// TwinCAT 3 PLC project GmdPlc
// ProgramVersion: 3.1.4022.3
// libraries:
//   L2SI Vacuum Library, * (SLAC)
//   LCLS General, * (SLAC)
//   Tc2_Standard, * (Beckhoff Automation GmbH)
//   Tc2_System, * (Beckhoff Automation GmbH)
//   Tc2_Utilities, * (Beckhoff Automation GmbH)
//   Tc3_Module, * (Beckhoff Automation GmbH)
// project tree:
//   GVLs/ GVL_GMD.TcGVL, GVL_VARIABLES.TcGVL
//   / PlcTask.TcTTO
//   POUs/ MAIN.TcPOU, PRG_DIAGNOSTIC.TcPOU, PRG_GMD.TcPOU
// real-time tasks:
//   TASK PlcTask: cycle T#10ms, priority 20, ADS port 350
//   TASK SimTask: cycle T#5ms, priority 21, ADS port 351
// I/O:
//   DEVICE =+-EK1100_00_00-CPU/EtherCAT1, AmsNetId 5.56.6.154.2.1
//     =+-EK1100_00_00 [EK1100 EtherCAT Coupler (2A E-Bus)]
//       =+-EK1110_00_08 [EK1110 EtherCAT extension]
//     =+-EL3174-02_04_08 [EL3174 4Ch. Ana. Input +/-10V Diff., +/-20mA SingleEnded, 16 Bit]
//     =+-ES9187_02_13 [EL9187 Potential Connection, 8 x Ground]
//     =+-ES9187_02_09 [EL9187 Potential Connection, 8 x Ground]
//     =+-ES9187_01_13 [EL9187 Potential Connection, 8 x Ground]
//     =+-ES9187_01_08 [EL9187 Potential Connection, 8 x Ground]
//     =+-ES9187_01_03 [EL9187 Potential Connection, 8 x Ground]
//     =+-ES9184_04_14 [EL9184 Potential Connection, 8 x 24V, 8 x Ground]
//     =+-ES9184_00_05 [EL9184 Potential Connection, 8 x 24V, 8 x Ground]
//     =+-ES9070_04_12 [EL9070 Shield terminal]
//     =+-ES9070_04_09 [EL9070 Shield terminal]
//     =+-ES9070_04_04 [EL9070 Shield terminal]
//     =+-ES9070_00_03 [EL9070 Shield terminal]
//     =+-ES7041_04_01 [EL7041 1Ch. Stepper motor output stage (50V, 5A)]
//     =+-ES4004_04_05 [EL4004 4Ch. Ana. Output 0-10V, 12bit]
//     =+-ES3202_04_10 [EL3202 2Ch. Ana. Input PT100 (RTD)]
//     =+-ES3068_01_14 [EL3068 8Ch. Ana. Input 0-10V]
//     =+-ES3068_01_12 [EL3068 8Ch. Ana. Input 0-10V]
//     =+-ES3068_01_09 [EL3068 8Ch. Ana. Input 0-10V]
//     =+-ES3068_01_07 [EL3068 8Ch. Ana. Input 0-10V]
//     =+-ES3068_01_04 [EL3068 8Ch. Ana. Input 0-10V]
//     =+-ES3068_01_02 [EL3068 8Ch. Ana. Input 0-10V]
//     =+-ES3064_04_11 [EL3064 4Ch. Ana. Input 0-10V]
//     =+-ES3064_00_02 [EL3064 4Ch. Ana. Input 0-10V]
//     =+-ES2088_02_14 [EL2088 8Ch. Dig. Output 24V, 0.5A, switching to negative]
//     =+-ES2088_02_10 [EL2088 8Ch. Dig. Output 24V, 0.5A, switching to negative]
//     =+-ES2008_04_15 [EL2008 8Ch. Dig. Output 24V, 0.5A]
//     =+-ES2008_00_06 [EL2008 8Ch. Dig. Output 24V, 0.5A]
//     =+-ES2004_04_07 [EL2004 4Ch. Dig. Output 24V, 0.5A]
//     =+-ES2004_04_06 [EL2004 4Ch. Dig. Output 24V, 0.5A]
//     =+-ES2004_02_05 [EL2004 4Ch. Dig. Output 24V, 0.5A]
//     =+-ES2004_02_02 [EL2004 4Ch. Dig. Output 24V, 0.5A]
//     =+-ES1088_02_15 [EL1088 8Ch. Dig. Input 24V, 3ms, negative]
//     =+-ES1088_02_12 [EL1088 8Ch. Dig. Input 24V, 3ms, negative]
//     =+-ES1088_02_11 [EL1088 8Ch. Dig. Input 24V, 3ms, negative]
//     =+-ES1088_02_08 [EL1088 8Ch. Dig. Input 24V, 3ms, negative]
//     =+-ES1008_04_13 [EL1008 8Ch. Dig. Input 24V, 3ms]
//     =+-ES1008_00_04 [EL1008 8Ch. Dig. Input 24V, 3ms]
//     =+-ES1004_02_06 [EL1004 4Ch. Dig. Input 24V, 3ms]
//     =+-ES1004_02_04 [EL1004 4Ch. Dig. Input 24V, 3ms]
//     =+-ES1004_02_03 [EL1004 4Ch. Dig. Input 24V, 3ms]
//     =+-ES1004_02_01 [EL1004 4Ch. Dig. Input 24V, 3ms]
//     =+-EL9400_02_07 [EL9400 E-Bus Power Supplier]
//     =+-EL2794_04_16 [EL2794 4Ch. Dig. Output 24V AC/DC, 2A, short-circuit-proof]
//     =+-EL2794_04_02 [EL2794 4Ch. Dig. Output 24V AC/DC, 2A, short-circuit-proof]
//     =+-EL2794_01_15 [EL2794 4Ch. Dig. Output 24V AC/DC, 2A, short-circuit-proof]
//     =+-EL2794_01_11 [EL2794 4Ch. Dig. Output 24V AC/DC, 2A, short-circuit-proof]
//     =+-EL2794_01_10 [EL2794 4Ch. Dig. Output 24V AC/DC, 2A, short-circuit-proof]
//     =+-EL2794_01_06 [EL2794 4Ch. Dig. Output 24V AC/DC, 2A, short-circuit-proof]
//     =+-EL2794_01_05 [EL2794 4Ch. Dig. Output 24V AC/DC, 2A, short-circuit-proof]
//     =+-EL2794_01_01 [EL2794 4Ch. Dig. Output 24V AC/DC, 2A, short-circuit-proof]
//     =+-EL2794_00_07 [EL2794 4Ch. Dig. Output 24V AC/DC, 2A, short-circuit-proof]
//     =+-EL1004_04_03 [EL1004 4Ch. Dig. Input 24V, 3ms]
//     =+-EK1110_04_17 [EK1110 EtherCAT extension]
//   DEVICE SimDevice 2 (EtherCAT Simulation), AmsNetId 5.45.6.154.3.1
//     =+-EK1100_00_00 // EK1100-0000-0018
//     =+-EK1110_00_08 // EK1110-0000-0017
//     =+-EL3174-02_04_08 // EL3174-0000-0016
//     =+-ES7041_04_01 // EL7041-0000-0025
//     =+-ES4004_04_05 // EL4004-0000-0020
//     =+-ES3202_04_10 // EL3202-0000-0022
//     =+-ES3068_01_14 // EL3068-0000-0020
//     =+-ES3068_01_12 // EL3068-0000-0020
//     =+-ES3068_01_09 // EL3068-0000-0020
//     =+-ES3068_01_07 // EL3068-0000-0020
//     =+-ES3068_01_04 // EL3068-0000-0020
//     =+-ES3068_01_02 // EL3068-0000-0020
//     =+-ES3064_04_11 // EL3064-0000-0020
//     =+-ES3064_00_02 // EL3064-0000-0020
//     =+-ES2088_02_14 // EL2088-0000-0018
//     =+-ES2088_02_10 // EL2088-0000-0018
//     =+-ES2008_04_15 // EL2008-0000-0018
//     =+-ES2008_00_06 // EL2008-0000-0018
//     =+-ES2004_04_07 // EL2004-0000-0018
//     =+-ES2004_04_06 // EL2004-0000-0018
//     =+-ES2004_02_05 // EL2004-0000-0018
//     =+-ES2004_02_02 // EL2004-0000-0018
//     =+-ES1088_02_15 // EL1088-0000-0018
//     =+-ES1088_02_12 // EL1088-0000-0018
//     =+-ES1088_02_11 // EL1088-0000-0018
//     =+-ES1088_02_08 // EL1088-0000-0018
//     =+-ES1008_04_13 // EL1008-0000-0018
//     =+-ES1008_00_04 // EL1008-0000-0018
//     =+-ES1004_02_06 // EL1004-0000-0019
//     =+-ES1004_02_04 // EL1004-0000-0019
//     =+-ES1004_02_03 // EL1004-0000-0019
//     =+-ES1004_02_01 // EL1004-0000-0019
//     =+-EL2794_04_16 // EL2794-0000-0016
//     =+-EL2794_04_02 // EL2794-0000-0016
//     =+-EL2794_01_15 // EL2794-0000-0016
//     =+-EL2794_01_11 // EL2794-0000-0016
//     =+-EL2794_01_10 // EL2794-0000-0016
//     =+-EL2794_01_06 // EL2794-0000-0016
//     =+-EL2794_01_05 // EL2794-0000-0016
//     =+-EL2794_01_01 // EL2794-0000-0016
//     =+-EL2794_00_07 // EL2794-0000-0016
//     =+-EL1004_04_03 // EL1004-0000-0019
//     =+-EK1110_04_17 // EK1110-0000-0017
// variable links:
//   GmdPlc/GmdPlc Instance <-> =+-EK1100_00_00-CPU/EtherCAT1/=+-EL1004_04_03
//     PlcTask Inputs/GVL_GMD.fb_EM1K0_GMD_PRT_40.i_xAlarmOK <-> Channel 2/Input
//     PlcTask Inputs/GVL_GMD.fb_EM1K0_GMD_PRT_40.i_xIsRun <-> Channel 1/Input
//   GmdPlc/GmdPlc Instance <-> =+-EK1100_00_00-CPU/EtherCAT1/=+-EL2794_01_01
//     PlcTask Outputs/GVL_GMD.fb_EM1K0_GMD_GCC_10.q_xHV_DIS <-> Channel 1/Output
//     PlcTask Outputs/GVL_GMD.fb_EM1K0_GMD_GCC_20.q_xHV_DIS <-> Channel 2/Output
//     PlcTask Outputs/GVL_GMD.fb_EM1K0_GMD_GCC_30.q_xHV_DIS <-> Channel 3/Output
//   GmdPlc/GmdPlc Instance <-> =+-EK1100_00_00-CPU/EtherCAT1/=+-EL2794_01_05
//     PlcTask Outputs/GVL_GMD.fb_EM1K0_GMD_GCC_40.q_xHV_DIS <-> Channel 2/Output
//   GmdPlc/GmdPlc Instance <-> =+-EK1100_00_00-CPU/EtherCAT1/=+-EL2794_01_06
//     PlcTask Outputs/GVL_GMD.fb_EM1K0_GMD_GCC_50.q_xHV_DIS <-> Channel 1/Output
//     PlcTask Outputs/GVL_GMD.fb_EM1K0_GMD_GCC_60.q_xHV_DIS <-> Channel 2/Output
//   GmdPlc/GmdPlc Instance <-> =+-EK1100_00_00-CPU/EtherCAT1/=+-EL2794_01_10
//     PlcTask Outputs/GVL_GMD.fb_EM1K0_GMD_GCC_70.q_xHV_DIS <-> Channel 1/Output
//   GmdPlc/GmdPlc Instance <-> =+-EK1100_00_00-CPU/EtherCAT1/=+-EL2794_04_02
//     PlcTask Outputs/GVL_GMD.fb_EM1K0_GMD_PRT_40.q_xRemote <-> Channel 2/Output
//     PlcTask Outputs/GVL_GMD.fb_EM1K0_GMD_PRT_40.q_xRunDo <-> Channel 1/Output
//   GmdPlc/GmdPlc Instance <-> =+-EK1100_00_00-CPU/EtherCAT1/=+-ES1004_02_01
//     PlcTask Inputs/GVL_GMD.fb_EM1K0_GMD_VRC_10.i_xClsLS <-> Channel 2/Input
//     PlcTask Inputs/GVL_GMD.fb_EM1K0_GMD_VRC_20.i_xClsLS <-> Channel 4/Input
//     PlcTask Inputs/GVL_GMD.fb_EM1K0_GMD_VRC_10.i_xOpnLS <-> Channel 1/Input
//     PlcTask Inputs/GVL_GMD.fb_EM1K0_GMD_VRC_20.i_xOpnLS <-> Channel 3/Input
//   GmdPlc/GmdPlc Instance <-> =+-EK1100_00_00-CPU/EtherCAT1/=+-ES1004_02_03
//     PlcTask Inputs/GVL_GMD.fb_EM1K0_GMD_VRC_30.i_xClsLS <-> Channel 2/Input
//     PlcTask Inputs/GVL_GMD.fb_EM1K0_GMD_VRC_30.i_xOpnLS <-> Channel 1/Input
//   GmdPlc/GmdPlc Instance <-> =+-EK1100_00_00-CPU/EtherCAT1/=+-ES1004_02_04
//     PlcTask Inputs/GVL_GMD.fb_EM1K0_GMD_VRC_50.i_xClsLS <-> Channel 2/Input
//     PlcTask Inputs/GVL_GMD.fb_EM1K0_GMD_VRC_60.i_xClsLS <-> Channel 4/Input
//     PlcTask Inputs/GVL_GMD.fb_EM1K0_GMD_VRC_50.i_xOpnLS <-> Channel 1/Input
//     PlcTask Inputs/GVL_GMD.fb_EM1K0_GMD_VRC_60.i_xOpnLS <-> Channel 3/Input
//   GmdPlc/GmdPlc Instance <-> =+-EK1100_00_00-CPU/EtherCAT1/=+-ES1004_02_06
//     PlcTask Inputs/GVL_GMD.fb_EM1K0_GMD_VRC_70.i_xClsLS <-> Channel 2/Input
//     PlcTask Inputs/GVL_GMD.fb_EM1K0_GMD_VRC_70.i_xOpnLS <-> Channel 1/Input
//   GmdPlc/GmdPlc Instance <-> =+-EK1100_00_00-CPU/EtherCAT1/=+-ES1088_02_08
//     PlcTask Inputs/GVL_GMD.fb_EM1K0_GMD_PTM_10.i_xAtSpd <-> Channel 1/Input
//     PlcTask Inputs/GVL_GMD.fb_EM1K0_GMD_PTM_20.i_xAtSpd <-> Channel 3/Input
//     PlcTask Inputs/GVL_GMD.fb_EM1K0_GMD_PTM_10.i_xFault <-> Channel 2/Input
//     PlcTask Inputs/GVL_GMD.fb_EM1K0_GMD_PTM_20.i_xFault <-> Channel 4/Input
//   GmdPlc/GmdPlc Instance <-> =+-EK1100_00_00-CPU/EtherCAT1/=+-ES1088_02_11
//     PlcTask Inputs/GVL_GMD.fb_EM1K0_GMD_PTM_30.i_xAtSpd <-> Channel 1/Input
//     PlcTask Inputs/GVL_GMD.fb_EM1K0_GMD_PTM_40.i_xAtSpd <-> Channel 3/Input
//     PlcTask Inputs/GVL_GMD.fb_EM1K0_GMD_PTM_30.i_xFault <-> Channel 2/Input
//     PlcTask Inputs/GVL_GMD.fb_EM1K0_GMD_PTM_40.i_xFault <-> Channel 4/Input
//   GmdPlc/GmdPlc Instance <-> =+-EK1100_00_00-CPU/EtherCAT1/=+-ES1088_02_12
//     PlcTask Inputs/GVL_GMD.fb_EM1K0_GMD_PTM_50.i_xAtSpd <-> Channel 1/Input
//     PlcTask Inputs/GVL_GMD.fb_EM1K0_GMD_PTM_60.i_xAtSpd <-> Channel 3/Input
//     PlcTask Inputs/GVL_GMD.fb_EM1K0_GMD_PTM_50.i_xFault <-> Channel 2/Input
//     PlcTask Inputs/GVL_GMD.fb_EM1K0_GMD_PTM_60.i_xFault <-> Channel 4/Input
//   GmdPlc/GmdPlc Instance <-> =+-EK1100_00_00-CPU/EtherCAT1/=+-ES1088_02_15
//     PlcTask Inputs/GVL_GMD.fb_EM1K0_GMD_PTM_70.i_xAtSpd <-> Channel 1/Input
//     PlcTask Inputs/GVL_GMD.fb_EM1K0_GMD_PTM_70.i_xFault <-> Channel 2/Input
//   GmdPlc/GmdPlc Instance <-> =+-EK1100_00_00-CPU/EtherCAT1/=+-ES2004_02_02
//     PlcTask Outputs/GVL_GMD.fb_EM1K0_GMD_VRC_10.q_xOPN_DO <-> Channel 1/Output
//     PlcTask Outputs/GVL_GMD.fb_EM1K0_GMD_VRC_20.q_xOPN_DO <-> Channel 2/Output
//     PlcTask Outputs/GVL_GMD.fb_EM1K0_GMD_VRC_30.q_xOPN_DO <-> Channel 3/Output
//   GmdPlc/GmdPlc Instance <-> =+-EK1100_00_00-CPU/EtherCAT1/=+-ES2004_02_05
//     PlcTask Outputs/GVL_GMD.fb_EM1K0_GMD_VRC_50.q_xOPN_DO <-> Channel 1/Output
//     PlcTask Outputs/GVL_GMD.fb_EM1K0_GMD_VRC_60.q_xOPN_DO <-> Channel 2/Output
//     PlcTask Outputs/GVL_GMD.fb_EM1K0_GMD_VRC_70.q_xOPN_DO <-> Channel 3/Output
//   GmdPlc/GmdPlc Instance <-> =+-EK1100_00_00-CPU/EtherCAT1/=+-ES2088_02_10
//     PlcTask Outputs/GVL_GMD.fb_EM1K0_GMD_PTM_{10..40 step 10}.q_RunDO <-> Channel {1..4}/Output  (4 links)
//   GmdPlc/GmdPlc Instance <-> =+-EK1100_00_00-CPU/EtherCAT1/=+-ES2088_02_14
//     PlcTask Outputs/GVL_GMD.fb_EM1K0_GMD_PTM_50.q_RunDO <-> Channel 1/Output
//     PlcTask Outputs/GVL_GMD.fb_EM1K0_GMD_PTM_60.q_RunDO <-> Channel 2/Output
//     PlcTask Outputs/GVL_GMD.fb_EM1K0_GMD_PTM_70.q_RunDO <-> Channel 3/Output
//   GmdPlc/GmdPlc Instance <-> =+-EK1100_00_00-CPU/EtherCAT1/=+-ES3068_01_02
//     PlcTask Inputs/GVL_GMD.fb_EM1K0_GMD_GCC_10.i_iPRESS_R <-> AI Standard Channel 1/Value
//     PlcTask Inputs/GVL_GMD.fb_EM1K0_GMD_GCC_20.i_iPRESS_R <-> AI Standard Channel 3/Value
//     PlcTask Inputs/GVL_GMD.fb_EM1K0_GMD_GCC_30.i_iPRESS_R <-> AI Standard Channel 5/Value
//   GmdPlc/GmdPlc Instance <-> =+-EK1100_00_00-CPU/EtherCAT1/=+-ES3068_01_04
//     PlcTask Inputs/GVL_GMD.fb_EM1K0_GMD_GCC_40.i_iPRESS_R <-> AI Standard Channel 3/Value
//     PlcTask Inputs/GVL_GMD.fb_EM1K0_GMD_GPI_10.i_iPRESS_R <-> AI Standard Channel 6/Value
//     PlcTask Inputs/GVL_GMD.fb_EM1K0_GMD_GPI_40.i_iPRESS_R <-> AI Standard Channel 5/Value
//   GmdPlc/GmdPlc Instance <-> =+-EK1100_00_00-CPU/EtherCAT1/=+-ES3068_01_07
//     PlcTask Inputs/GVL_GMD.fb_EM1K0_GMD_GCC_50.i_iPRESS_R <-> AI Standard Channel 1/Value
//     PlcTask Inputs/GVL_GMD.fb_EM1K0_GMD_GCC_60.i_iPRESS_R <-> AI Standard Channel 3/Value
//     PlcTask Inputs/GVL_GMD.fb_EM1K0_GMD_GPI_70.i_iPRESS_R <-> AI Standard Channel 6/Value
//   GmdPlc/GmdPlc Instance <-> =+-EK1100_00_00-CPU/EtherCAT1/=+-ES3068_01_09
//     PlcTask Inputs/GVL_GMD.fb_EM1K0_GMD_GCC_70.i_iPRESS_R <-> AI Standard Channel 1/Value
//   GmdSim/GmdSim Instance <-> SimDevice 2 (EtherCAT Simulation)/=+-EL2794_01_01
//     SimTask Inputs/GVL_GMD.st_EM1K0_GMD_GCC_10.i_xHvOn <-> Channel 1/Output
//     SimTask Inputs/GVL_GMD.st_EM1K0_GMD_GCC_20.i_xHvOn <-> Channel 2/Output
//     SimTask Inputs/GVL_GMD.st_EM1K0_GMD_GCC_30.i_xHvOn <-> Channel 3/Output
//   GmdSim/GmdSim Instance <-> SimDevice 2 (EtherCAT Simulation)/=+-EL2794_01_05
//     SimTask Inputs/GVL_GMD.st_EM1K0_GMD_GCC_40.i_xHvOn <-> Channel 2/Output
//   GmdSim/GmdSim Instance <-> SimDevice 2 (EtherCAT Simulation)/=+-EL2794_01_06
//     SimTask Inputs/GVL_GMD.st_EM1K0_GMD_GCC_50.i_xHvOn <-> Channel 1/Output
//     SimTask Inputs/GVL_GMD.st_EM1K0_GMD_GCC_60.i_xHvOn <-> Channel 2/Output
//   GmdSim/GmdSim Instance <-> SimDevice 2 (EtherCAT Simulation)/=+-EL2794_01_10
//     SimTask Inputs/GVL_GMD.st_EM1K0_GMD_GCC_70.i_xHvOn <-> Channel 1/Output
//   GmdSim/GmdSim Instance <-> SimDevice 2 (EtherCAT Simulation)/=+-ES1004_02_01
//     SimTask Outputs/GVL_GMD.st_EM1K0_GMD_VRC_10.q_xClsLS <-> Channel 2/Input
//     SimTask Outputs/GVL_GMD.st_EM1K0_GMD_VRC_20.q_xClsLS <-> Channel 4/Input
//     SimTask Outputs/GVL_GMD.st_EM1K0_GMD_VRC_10.q_xOpnLS <-> Channel 1/Input
//     SimTask Outputs/GVL_GMD.st_EM1K0_GMD_VRC_20.q_xOpnLS <-> Channel 3/Input
//   GmdSim/GmdSim Instance <-> SimDevice 2 (EtherCAT Simulation)/=+-ES1004_02_03
//     SimTask Outputs/GVL_GMD.st_EM1K0_GMD_VRC_30.q_xClsLS <-> Channel 2/Input
//     SimTask Outputs/GVL_GMD.st_EM1K0_GMD_VRC_30.q_xOpnLS <-> Channel 1/Input
//   GmdSim/GmdSim Instance <-> SimDevice 2 (EtherCAT Simulation)/=+-ES1004_02_04
//     SimTask Outputs/GVL_GMD.st_EM1K0_GMD_VRC_50.q_xClsLS <-> Channel 2/Input
//     SimTask Outputs/GVL_GMD.st_EM1K0_GMD_VRC_60.q_xClsLS <-> Channel 4/Input
//     SimTask Outputs/GVL_GMD.st_EM1K0_GMD_VRC_50.q_xOpnLS <-> Channel 1/Input
//     SimTask Outputs/GVL_GMD.st_EM1K0_GMD_VRC_60.q_xOpnLS <-> Channel 3/Input
//   GmdSim/GmdSim Instance <-> SimDevice 2 (EtherCAT Simulation)/=+-ES1004_02_06
//     SimTask Outputs/GVL_GMD.st_EM1K0_GMD_VRC_70.q_xClsLS <-> Channel 2/Input
//     SimTask Outputs/GVL_GMD.st_EM1K0_GMD_VRC_70.q_xOpnLS <-> Channel 1/Input
//   GmdSim/GmdSim Instance <-> SimDevice 2 (EtherCAT Simulation)/=+-ES2004_02_02
//     SimTask Inputs/GVL_GMD.st_EM1K0_GMD_VRC_10.i_xSol <-> Channel 1/Output
//     SimTask Inputs/GVL_GMD.st_EM1K0_GMD_VRC_20.i_xSol <-> Channel 2/Output
//     SimTask Inputs/GVL_GMD.st_EM1K0_GMD_VRC_30.i_xSol <-> Channel 3/Output
//   GmdSim/GmdSim Instance <-> SimDevice 2 (EtherCAT Simulation)/=+-ES2004_02_05
//     SimTask Inputs/GVL_GMD.st_EM1K0_GMD_VRC_50.i_xSol <-> Channel 1/Output
//     SimTask Inputs/GVL_GMD.st_EM1K0_GMD_VRC_60.i_xSol <-> Channel 2/Output
//     SimTask Inputs/GVL_GMD.st_EM1K0_GMD_VRC_70.i_xSol <-> Channel 3/Output
//   GmdSim/GmdSim Instance <-> SimDevice 2 (EtherCAT Simulation)/=+-ES3068_01_02
//     SimTask Outputs/GVL_GMD.st_EM1K0_GMD_GCC_10.q_iRawPress <-> AI Standard Channel 1/Value
//     SimTask Outputs/GVL_GMD.st_EM1K0_GMD_GCC_20.q_iRawPress <-> AI Standard Channel 3/Value
//     SimTask Outputs/GVL_GMD.st_EM1K0_GMD_GCC_30.q_iRawPress <-> AI Standard Channel 5/Value
//   GmdSim/GmdSim Instance <-> SimDevice 2 (EtherCAT Simulation)/=+-ES3068_01_04
//     SimTask Outputs/GVL_GMD.st_EM1K0_GMD_GCC_40.q_iRawPress <-> AI Standard Channel 3/Value
//     SimTask Outputs/GVL_GMD.st_EM1K0_GMD_GPI_10.q_iRawPress <-> AI Standard Channel 6/Value
//     SimTask Outputs/GVL_GMD.st_EM1K0_GMD_GPI_40.q_iRawPress <-> AI Standard Channel 5/Value
//   GmdSim/GmdSim Instance <-> SimDevice 2 (EtherCAT Simulation)/=+-ES3068_01_07
//     SimTask Outputs/GVL_GMD.st_EM1K0_GMD_GCC_50.q_iRawPress <-> AI Standard Channel 1/Value
//     SimTask Outputs/GVL_GMD.st_EM1K0_GMD_GCC_60.q_iRawPress <-> AI Standard Channel 3/Value
//     SimTask Outputs/GVL_GMD.st_EM1K0_GMD_GPI_70.q_iRawPress <-> AI Standard Channel 6/Value
//   GmdSim/GmdSim Instance <-> SimDevice 2 (EtherCAT Simulation)/=+-ES3068_01_09
//     SimTask Outputs/GVL_GMD.st_EM1K0_GMD_GCC_70.q_iRawPress <-> AI Standard Channel 1/Value

CONFIGURATION GmdPlc
    RESOURCE PLC ON TwinCAT3
        TASK PlcTask(INTERVAL := T#10ms, PRIORITY := 20);
        PROGRAM MAIN WITH PlcTask : MAIN;
    END_RESOURCE
END_CONFIGURATION

// ---- GVLs/GVL_GMD.TcGVL
VAR_GLOBAL

// FB_MKS317

{attribute 'pytmc' := ' pv: EM1K0:GMD:GPI:10 '}
fb_EM1K0_GMD_GPI_10 : FB_MKS317;
{attribute 'pytmc' := ' pv: EM1K0:GMD:GPI:40 '}
fb_EM1K0_GMD_GPI_40 : FB_MKS317;
{attribute 'pytmc' := ' pv: EM1K0:GMD:GPI:70 '}
fb_EM1K0_GMD_GPI_70 : FB_MKS317;

// FB_PTM_TwisTorr

{attribute 'pytmc' := ' pv: EM1K0:GMD:PTM:10 '}
fb_EM1K0_GMD_PTM_10 : FB_PTM_TwisTorr;
{attribute 'pytmc' := ' pv: EM1K0:GMD:PTM:20 '}
fb_EM1K0_GMD_PTM_20 : FB_PTM_TwisTorr;
{attribute 'pytmc' := ' pv: EM1K0:GMD:PTM:30 '}
fb_EM1K0_GMD_PTM_30 : FB_PTM_TwisTorr;
{attribute 'pytmc' := ' pv: EM1K0:GMD:PTM:40 '}
fb_EM1K0_GMD_PTM_40 : FB_PTM_TwisTorr;
{attribute 'pytmc' := ' pv: EM1K0:GMD:PTM:50 '}
fb_EM1K0_GMD_PTM_50 : FB_PTM_TwisTorr;
{attribute 'pytmc' := ' pv: EM1K0:GMD:PTM:60 '}
fb_EM1K0_GMD_PTM_60 : FB_PTM_TwisTorr;
{attribute 'pytmc' := ' pv: EM1K0:GMD:PTM:70 '}
fb_EM1K0_GMD_PTM_70 : FB_PTM_TwisTorr;

// FB_VRC

{attribute 'pytmc' := ' pv: EM1K0:GMD:VRC:10 '}
fb_EM1K0_GMD_VRC_10 : FB_VRC;
{attribute 'pytmc' := ' pv: EM1K0:GMD:VRC:20 '}
fb_EM1K0_GMD_VRC_20 : FB_VRC;
{attribute 'pytmc' := ' pv: EM1K0:GMD:VRC:30 '}
fb_EM1K0_GMD_VRC_30 : FB_VRC;
{attribute 'pytmc' := ' pv: EM1K0:GMD:VRC:50 '}
fb_EM1K0_GMD_VRC_50 : FB_VRC;
{attribute 'pytmc' := ' pv: EM1K0:GMD:VRC:60 '}
fb_EM1K0_GMD_VRC_60 : FB_VRC;
{attribute 'pytmc' := ' pv: EM1K0:GMD:VRC:70 '}
fb_EM1K0_GMD_VRC_70 : FB_VRC;

// FB_MKS422

{attribute 'pytmc' := ' pv: EM1K0:GMD:GCC:10 '}
fb_EM1K0_GMD_GCC_10 : FB_MKS422;
{attribute 'pytmc' := ' pv: EM1K0:GMD:GCC:20 '}
fb_EM1K0_GMD_GCC_20 : FB_MKS422;
{attribute 'pytmc' := ' pv: EM1K0:GMD:GCC:30 '}
fb_EM1K0_GMD_GCC_30 : FB_MKS422;
{attribute 'pytmc' := ' pv: EM1K0:GMD:GCC:40 '}
fb_EM1K0_GMD_GCC_40 : FB_MKS422;
{attribute 'pytmc' := ' pv: EM1K0:GMD:GCC:50 '}
fb_EM1K0_GMD_GCC_50 : FB_MKS422;
{attribute 'pytmc' := ' pv: EM1K0:GMD:GCC:60 '}
fb_EM1K0_GMD_GCC_60 : FB_MKS422;
{attribute 'pytmc' := ' pv: EM1K0:GMD:GCC:70 '}
fb_EM1K0_GMD_GCC_70 : FB_MKS422;

// FB_EbaraEVA

{attribute 'pytmc' := ' pv: EM1K0:GMD:PRT:40 '}
fb_EM1K0_GMD_PRT_40 : FB_EbaraEVA;

END_VAR

// ---- GVLs/GVL_VARIABLES.TcGVL
VAR_GLOBAL
	xSystemOverrideMode : BOOL; (* Global system override for the prototype section*)
END_VAR

// ---- POUs/MAIN.TcPOU
PROGRAM MAIN
VAR
END_VAR

PRG_DIAGNOSTIC();
PRG_GMD();

END_PROGRAM

// ---- POUs/PRG_DIAGNOSTIC.TcPOU
PROGRAM PRG_DIAGNOSTIC
VAR
   fbTime : FB_LocalSystemTime := ( bEnable := TRUE, dwCycle := 1 );
   logTimer : TON := ( IN := TRUE, PT := T#1000ms );

   plcName : STRING[15];

   {attribute 'pytmc' := ' pv: simHeartbeat '}
   simHeartbeat AT %I* : UINT := 0;
   {attribute 'pytmc' := ' pv: plcHeartbeat '}
   plcHeartbeat : UDINT := 0;
   {attribute 'pytmc' := ' pv: plcInfo '}
   plcInfo : STRING[40];
   {attribute 'pytmc' := ' pv: plcLocalTime '}
   plcLocalTime : STRING[25];
   
END_VAR

plcHeartbeat := plcHeartbeat + 1;
IF plcHeartbeat > 4294967000
   THEN plcHeartbeat := 0;
END_IF

// get timestamp as string every second
fbTime();
logTimer( IN := fbTime.bValid );
IF logTimer.Q THEN
   logTimer( IN := FALSE ); logTimer( IN := fbTime.bValid );
   plcLocalTime := SYSTEMTIME_TO_STRING(fbTime.systemTime);
END_IF

// make an info string
plcName := 'Prototype PLC: ';
plcInfo := CONCAT(plcName, plcLocalTime);

END_PROGRAM

// ---- POUs/PRG_GMD.TcPOU
PROGRAM PRG_GMD
VAR
END_VAR


// FB_MKS317

fb_EM1K0_GMD_GPI_10(PG=>);
fb_EM1K0_GMD_GPI_40(PG=>);
fb_EM1K0_GMD_GPI_70(PG=>);

// FB_PTM_TwisTorr

fb_EM1K0_GMD_PTM_10(i_xExtILKOk := TRUE);
fb_EM1K0_GMD_PTM_20(i_xExtILKOk := TRUE);
fb_EM1K0_GMD_PTM_30(i_xExtILKOk := TRUE);
fb_EM1K0_GMD_PTM_40(i_xExtILKOk := TRUE);
fb_EM1K0_GMD_PTM_50(i_xExtILKOk := TRUE);
fb_EM1K0_GMD_PTM_60(i_xExtILKOk := TRUE);
fb_EM1K0_GMD_PTM_70(i_xExtILKOk := TRUE);

// FB_VRC

fb_EM1K0_GMD_VRC_10(i_xExtILK_OK := TRUE, i_xOverrideMode := xSystemOverrideMode);
fb_EM1K0_GMD_VRC_20(i_xExtILK_OK := TRUE, i_xOverrideMode := xSystemOverrideMode);
fb_EM1K0_GMD_VRC_30(i_xExtILK_OK := TRUE, i_xOverrideMode := xSystemOverrideMode);
fb_EM1K0_GMD_VRC_50(i_xExtILK_OK := TRUE, i_xOverrideMode := xSystemOverrideMode);
fb_EM1K0_GMD_VRC_60(i_xExtILK_OK := TRUE, i_xOverrideMode := xSystemOverrideMode);
fb_EM1K0_GMD_VRC_70(i_xExtILK_OK := TRUE, i_xOverrideMode := xSystemOverrideMode);

// FB_MKS422

fb_EM1K0_GMD_GCC_10(PG := fb_EM1K0_GMD_GPI_10.PG);
fb_EM1K0_GMD_GCC_20(PG := fb_EM1K0_GMD_GPI_10.PG);
fb_EM1K0_GMD_GCC_30(PG := fb_EM1K0_GMD_GPI_10.PG);
fb_EM1K0_GMD_GCC_40(PG := fb_EM1K0_GMD_GPI_40.PG);
fb_EM1K0_GMD_GCC_50(PG := fb_EM1K0_GMD_GPI_70.PG);
fb_EM1K0_GMD_GCC_60(PG := fb_EM1K0_GMD_GPI_70.PG);
fb_EM1K0_GMD_GCC_70(PG := fb_EM1K0_GMD_GPI_70.PG);

// FB_EbaraEVA

fb_EM1K0_GMD_PRT_40(i_xExtIlkOK := TRUE);

END_PROGRAM
